(* Logix 5000 project; controller HPU_Part_Evac_Start 1769-L33ERM rev 30.11; software revision 30.01 *)

TASK MainTask (continuous, watchdog 500 ms) : MainProgram, Motion_Tools

MODULES
   Local : 1769-L33ERM (Compact 0, rev 30.11)
      Ecyl_1 : vendor 1 type 37 code 32 (Ethernet 192.168.1.21, rev 2.1, MotionSync RPI 1 ms, MotionDiagnostics RPI 1 ms)   // E Cylinder Station 1
      Ecyl_2 : vendor 1 type 37 code 32 (Ethernet 192.168.1.22, rev 2.1, MotionDiagnostics RPI 1 ms, MotionSync RPI 1 ms)   // E Cylinder Station 2
      Ecyl_4 : vendor 1 type 37 code 32 (Ethernet 192.168.1.24, rev 2.1, MotionSync RPI 1 ms, MotionDiagnostics RPI 1 ms)   // E Cylinder Station 4
      Ecyl_3 : vendor 1 type 37 code 32 (Ethernet 192.168.1.23, rev 2.1, MotionSync RPI 1 ms, MotionDiagnostics RPI 1 ms)   // E Cylinder Station 3
END_MODULES

TYPE Sequence1 :   // Sequence Start Conditions Met
STRUCT
   Perm : BOOL;   // Permissive to Advance
   Step : INT;   // Step Number
   Fault : BOOL;   // Fault
   Fault_Code : INT;   // Fault Code
   On : BOOL;   // Enabled
   StepMode : BOOL;   // Step Mode Enabled
   StepNext : BOOL;   // Next Step
   Status : STRING;   // Current Status
   Reset : BOOL;   // Reset Sequence
   Complete : BOOL;   // Sequence Complete [OS]
   PermLostStep : INT;   // Step where Permissive was Lost
   Home : BOOL;   // Sequence Actuators at Home
   StartCond : BOOL;   // Sequence Start Conditions Met
   HomeReq : BOOL;   // Sequence Home Request
   Step_Msg : STRING;   // Operator Message from Sequence
END_STRUCT
END_TYPE

TYPE Sequence_Ctrl :   // Sequence Start Conditions Met
STRUCT
   Perm : BOOL;   // Permissive to Advance
   Step : INT;   // Step Number
   Fault : BOOL;   // Fault
   Fault_Code : INT;   // Fault Code
   On : BOOL;   // Enabled
   StepMode : BOOL;   // Step Mode Enabled
   StepNext : BOOL;   // Next Step
   Status : STRING;   // Current Status
   Reset : BOOL;   // Reset Sequence
   Complete : BOOL;   // Sequence Complete [OS]
   PermLostStep : INT;   // Step where Permissive was Lost
   Home : BOOL;   // Sequence Actuators at Home
   StartCond : BOOL;   // Sequence Start Conditions Met
   HomeReq : BOOL;   // Sequence Home Request
   Step_Msg : STRING;   // Operator Message from Sequence
END_STRUCT
END_TYPE

VAR_GLOBAL   (* controller tags *)
   _Always_Off : BOOL;   // Always Off
   ai_Cylinder_Posn_Sta_1 : INT;   // Cylinder Position Station 1 Analog Input Raw Count Value
   ai_Cylinder_Posn_Sta_2 : INT;   // Cylinder Pressure Station 2 Analog Input Raw Count Value
   ai_Cylinder_Posn_Sta_3 : INT;   // Cylinder Pressure Station 3 Analog Input Raw Count Value
   ai_Cylinder_Posn_Sta_4 : INT;   // Cylinder Pressure Station 4 Analog Input Raw Count Value
   ai_Cylinder_Press_Sta_1 : INT;   // Cylinder Pressure Station 1 Analog Input Raw Count Value
   ai_Cylinder_Press_Sta_2 : INT;   // Cylinder Pressure Station 2 Analog Input Raw Count Value
   ai_Cylinder_Press_Sta_3 : INT;   // Cylinder Pressure Station 3 Analog Input Raw Count Value
   ai_Cylinder_Press_Sta_4 : INT;   // Cylinder Pressure Station 4 Analog Input Raw Count Value
   ao_Pressure_Relief_Out_Sta_1 : INT;   // Cylinder Relief Pressure Output Station 1 Analog Output Raw Count Value
   ao_Pressure_Relief_Out_Sta_2 : INT;   // Cylinder Relief Pressure Output Station 2 Analog Output Raw Count Value
   ao_Pressure_Relief_Out_Sta_3 : INT;   // Cylinder Relief Pressure Output Station 3 Analog Output Raw Count Value
   ao_Pressure_Relief_Out_Sta_4 : INT;   // Cylinder Relief Pressure Output Station 4 Analog Output Raw Count Value
   c_Ecyl_1_Auto_Exe_Inc : BOOL;   // Coil Ecylinder 1 Axis Auto Move (Incremental Move)
   c_MCR_On_Dly_PUL : BOOL;   // Coil MCR is On (1 Sec Delay) (250ms Pulse)
   c_Sld_Auto_Exe : BOOL;   // Coil Slide Auto Move (Absolute)
   c_Sld_Man_DS_Exe : BOOL;   // Coil Slide Axis Manual Move (Drive Screen)
   c_Sld_Man_PS_Cut : BOOL;   // Coil Slide Axis Manual Move Cut Position Pro Stich
   c_Sld_Man_PS_Grind : BOOL;   // Coil Slide Axis Manual Move Grind Position Pro Stich
   c_Sld_Man_PS_Grind_End : BOOL;   // Coil Slide Axis Manual Move Grind End Position Pro Stich
   c_Sld_Man_PS_Home : BOOL;   // Coil Slide Axis Manual Move Home Position Pro Stich
   c_Sld_Man_TR_End : BOOL;   // Coil Slide Axis Manual Move End Position Trheaded Rod
   c_Sld_Man_TR_Home : BOOL;   // Coil Slide Axis Manual Move Home Position Trheaded Rod
   c_Sld_Man_TR_Start : BOOL;   // Coil Slide Axis Manual Move Start Position Trheaded Rod
   c_Sld_Man_TR_Taper_Start : BOOL;   // Coil Slide Axis Manual Move Taper Start Position Trheaded Rod
   cntl_Mag_sld : MOTION_INSTRUCTION := (FLAGS := 570425344, DN := 1);   // Axes Sync Control
   cntl_Rot_UnSync : MOTION_INSTRUCTION := (FLAGS := 704643072, DN := 1, PC := 1);
   cntl_Sld_Air_Stop : MOTION_INSTRUCTION := (FLAGS := 33554432);
   cntl_Sld_Chng_Spd : MOTION_INSTRUCTION := (FLAGS := 570425344, DN := 1);
   cntl_Sld_Home : MOTION_INSTRUCTION := (FLAGS := 704643072, DN := 1, PC := 1, STATE := 17);   // Servo Control Slide Axis Home
   cntl_Sld_Off : MOTION_INSTRUCTION := (FLAGS := 570425344, DN := 1, STATUS := 2, STATE := 1);   // Servo Control Slide Axis Off
   cntl_Sld_On : MOTION_INSTRUCTION := (FLAGS := 570425344, DN := 1, STATE := 1);   // Servo Control Slide Axis On
   cntl_Sld_Reset : MOTION_INSTRUCTION := (FLAGS := 570425344, DN := 1, STATE := 1);   // Servo Control Slide Axis Fault Reset
   cntl_Sld_SD_Reset : MOTION_INSTRUCTION := (FLAGS := 33554432);   // Servo Control Slide Axis Shutdown Reset
   cntl_Sld_Stop : MOTION_INSTRUCTION := (FLAGS := 33554432);   // Motion Control Slide Axis Axis Stop
   cPV_Sld_Tpr_Vel : REAL := 0.033333335;   // Calculated slide velocity for tapered portion of thread.
   cPV_Sta_1_Cyl_Posn : REAL;   // Scaled Station 1 Stacking Cyclinder Position
   cPV_Sta_1_Cyl_Pressure : REAL;   // Scaled Station 1 Stacking Cyclinder Pressure
   cPV_Sta_2_Cyl_Posn : REAL;   // Scaled Station 2 Stacking Cyclinder Position
   cPV_Sta_2_Cyl_Pressure : REAL;   // Scaled Station 2 Stacking Cyclinder Position
   cPV_Sta_3_Cyl_Posn : REAL;   // Scaled Station 3 Stacking Cyclinder Position
   cPV_Sta_3_Cyl_Pressure : REAL;   // Scaled Station 3 Stacking Cyclinder Position
   cPV_Sta_4_Cyl_Posn : REAL;   // Scaled Station 4 Stacking Cyclinder Position
   cPV_Sta_4_Cyl_Pressure : REAL;   // Scaled Station 4 Stacking Cyclinder Position
   cSP_TR_Pitch : REAL := 5.0;   // Treaded Rod Pitch
   cSP_TR_Ratio : REAL := 1800.0;
   Drives_OK : BOOL := 1;   // All Drives OK
   ECyl_1 : AXIS_CIP_DRIVE;   // E Cylinder # 1
   ECyl_2 : AXIS_CIP_DRIVE;   // E Cylinder # 2
   Ecyl_3 : AXIS_CIP_DRIVE;
   Ecyl_4 : AXIS_CIP_DRIVE;
   hPB_All_Servo_On : BOOL;   // HMI Pushbutton All Servos On
   hPB_All_Servos_Off : BOOL;   // HMI Pushbutton All Servos OFF
   Hpb_Home : BOOL;   // HMI Pushbutton Machine Home
   hPB_MS_Hyd_Pump : BOOL;   // HMI PB Enable Hydraulic Pump
   hPB_Sld_AbsMv : BOOL;   // HMI Pushbutton Datum Bottom Axis Manual Move Absolute (From Drive Screen)
   hPB_Sld_Home : BOOL;   // HMI Pushbutton Slide Axis Home
   hPB_Sld_IncMv : BOOL;   // HMI Pushbutton Slide Axis Manual Move Incremental (From Drive Screen)
   hPB_Sld_MMv_PS_Cut : BOOL;   // HMI Pushbutton Slide Axis Pro Stich >>Move to Cut Position
   hPB_Sld_MMv_PS_Grind : BOOL;   // HMI Pushbutton Slide Axis Pro Stich >>Move to Grind Position
   hPB_Sld_MMv_PS_Grind_End : BOOL;   // HMI Pushbutton Slide Axis Pro Stich >>Move to Grind End Position
   hPB_Sld_MMv_PS_Home : BOOL;   // HMI Pushbutton Slide Axis Pro Stich >>Move to Home Position
   hPB_Sld_MMv_TR_End : BOOL;   // HMI Pushbutton Slide Axis Threaded Rod >>Move to End Position
   hPB_Sld_MMv_TR_Home : BOOL;   // HMI Pushbutton Slide Axis Threaded Rod >>Move to Home Position
   hPB_Sld_MMv_TR_Start : BOOL;   // HMI Pushbutton Slide Axis Threaded Rod >>Move to Start Position
   hPB_Sld_MMv_TR_Taper_Start : BOOL;   // HMI Pushbutton Slide Axis Threaded Rod >>Move to Taper Start Position
   hPB_Sld_Reset : BOOL;   // HMI Pushbutton Slide Axis Servo Reset
   hPB_Sld_ServoOff : BOOL;   // HMI Pushbutton Slide Axis Servo Axis Servo Off
   hPB_Sld_ServoOn : BOOL;   // HMI Pushbutton Slide Axis Servo Axis Servo On
   hPB_SV_Dump_Valve : BOOL;   // HMI PB Pressure Dump Solenoid Valve
   hPB_Sync_R_S : BOOL;   // Sync Rotary to Slide
   hPB_UnSync_R_S : BOOL;   // UnSync Rotary Axis from Slide
   hpl_Ecyl_1_Enabled : BOOL;   // E Cylinder 1 Enabled
   hpl_Ecyl_2_Enabled : BOOL;   // E Cylinder 2 Enabled
   hPL_PS_Active : BOOL;   // Pro-Stich Sequence Active
   hpv_Ecyl_1_Posn : REAL;   // E Cylinder 1 Position (mm)
   hpv_Ecyl_2_Posn : REAL;   // E Cylinder 2 Position (mm)
   hpv_Ecyl_3_Enabled : BOOL;   // E Cylinder 3 Enabled
   hpv_Ecyl_3_Posn : REAL;   // E Cylinder 3 Position (mm)
   hpv_Ecyl_4_Enabled : BOOL;   // E Cylinder 4 Enabled
   hpv_Ecyl_4_Posn : REAL;   // E Cylinder 4 Position (mm)
   hSP_Ecyl_1_DS_AbsMov : REAL := 10.0;   // HMI Setpoint Ecylinder 1 Axis (Drive Screen) Manual Absolute Move
   hSP_Ecyl_1_DS_IncMov : REAL := 20.0;   // HMI Setpoint Ecylinder 1 Axis (Drive Screen) Manual Incremental Move
   hSP_Ecyl_ManMove_Vel : REAL := 25.0;   // HMI Setpoint Ecylinder Axis Manual Move Velocity
   hSP_Ecyl_Pos_DB : REAL := 0.01;   // HMI Setpoint Ecylinder Positioning Deadband
   hSP_PS_Ecyl_1_Psp_Clear : REAL := 161.7784;   // HMI Setpoint Ecylinder 1 Clear of Stacking Cylinder Location
   hSP_PS_Ecyl_1_Psp_Home : REAL := 10.0;   // HMI Setpoint Ecylinder 1 HOME
   hSP_PS_Ecyl_1_Psp_Stacking : REAL := 166.4166;   // HMI Setpoint Ecylinder 1 Stacking Location
   hSP_PS_Ecyl_1_Psp_Unload : REAL := 158.5634;   // HMI Setpoint Ecylinder 1 Unload Location
   hSP_TR_Rot_Dir : DINT;
   hSP_TR_Sld_Psp_End : REAL := 100.0;   // Threaded Rod END Location Setpoint
   hSP_TR_Sld_Psp_Home : REAL := 10.0;   // Threaded Rod Home Position Setpoint
   hSP_TR_Sld_Psp_Start : REAL := 90.0;   // Threaded Rod START Position Setpoint
   hSP_TR_Sld_Psp_Taper_Start : REAL := 99.0;   // Threaded Rod Taper START Position Setpoint
   hSP_TR_TPM : REAL := 5.0;   // Treaded Rod Threads per Millimeter
   i_cr_Die_Position : BOOL;   // Die Position Sensor 1 = Die Closed
   i_cr_E_Stop : BOOL;   // Press Light Curtain and E Stop Input Relay Contacts
   i_cr_Pump_OL : BOOL;   // Hydraulic Pump Overload Contacts, NC
   i_cr_Pump_Running : BOOL;   // Hydraulic Pump running auxiliary contacts.
   i_cr_Stack_Done_Sta_1 : BOOL;   // Stack Done Station 1 signal from VAMCO
   i_cr_Stack_Done_Sta_2 : BOOL;   // Stack Done Station 2 signal from VAMCO
   i_cr_Stack_Done_Sta_3 : BOOL;   // Stack Done Station 3 signal from VAMCO
   i_cr_Stack_Done_Sta_4 : BOOL;   // Stack Done Station 4 signal from VAMCO
   i_pb_Cycle_Start : BOOL;   // Cycle Start Pushbutton Input
   i_pb_Cycle_Stop : BOOL;   // Cycle Stop Pushbutton Input
   i_pb_Reset : BOOL;   // Reset Pushbutton input
   IB_Man_Jog_Active : BOOL;   // Interface Bit used for Manual Jog Functions Starts Hydraulic Pump and Dump Valve
   IB_MS_Hyd_Pump : BOOL;   // Interface bit to run Hydraulic Pump in cycle.
   IB_PS_AMT_Sld : BOOL;   // Pro-Stich Auto Motion Trigger Slide Axis
   IB_PS_Loc_Ecyl_1_Clear : BOOL;   // Ecylinder 1 Location Bit Clear of Stacking Cylinder
   IB_PS_Loc_Ecyl_1_Home : BOOL := 1;   // Ecylinder 1 Location Bit Ecylinder 1 @ HOME
   IB_PS_Loc_Ecyl_1_Stacking : BOOL;   // Ecylinder 1 Location Bit Ecyl 1 @ Stacking
   IB_PS_Loc_Ecyl_1_Unload : BOOL;   // Ecylinder 1 Location Bit Ecylinder 1 @ Part Unload
   IB_SV_Dump_Valve : BOOL;   // Interface bit to trigger Dydraulic Pressure Dump Valve.
   IB_TR_AMT_Sld : BOOL;   // Threaded Rod Auto Motion Trigger Slide Axis
   IB_TR_Change_Speed : BOOL;   // Threaded Rod UnSync Axes
   IB_TR_Loc_Sld_End : BOOL;   // Threaded Rod Location Bit Slide @ END
   IB_TR_Loc_Sld_Home : BOOL := 1;   // Threaded Rod Location Bit Slide @ HOME
   IB_TR_Loc_Sld_Start : BOOL;   // Threaded Rod Location Bit Slide @ START
   IB_TR_Loc_Sld_Taper_Region : BOOL;   // Threaded Rod Location Bit Slide between Taper Start and END positions
   IB_TR_Loc_Sld_Taper_Start : BOOL;   // Threaded Rod Location Bit Slide at Taper Start position
   IB_TR_Sync_Axes : BOOL;   // Threaded Rod Sync Axes (Slave Rotate to Slide)
   IB_TR_UnSync_Axes : BOOL;   // Threaded Rod UnSync Axes
   M_Auto : BOOL;   // Machine in Auto Mode Sequence Cycle Start/Stop Active
   M_Manual : BOOL;   // Machine in Manual Mode, Outputs Controlled by HMI Buttons.
   M_Reset_Sum : BOOL;   // Machine Mode Reset_Sum
   MC_Sld_MAM : MOTION_INSTRUCTION := (FLAGS := 704643072, DN := 1, PC := 1);   // Motion Control Tag Slide Axis Motion Axis Move
   o_cr_Top_Stop : BOOL;   // Top Stop Relay Contacts to Press
   o_ms_Pump_Contactor : BOOL;   // Hydraulic Pump Contactor
   o_pl_Reset_Light : BOOL;   // Reset Pushbutton Light
   o_sv_Extend_Cyl_Sta_1 : BOOL;   // Extend Cylinder Station 1 Solenoid Valve
   o_sv_Extend_Cyl_Sta_2 : BOOL;   // Extend Cylinder Station 2 Solenoid Valve
   o_sv_Extend_Cyl_Sta_3 : BOOL;   // Extend Cylinder Station 3 Solenoid Valve
   o_sv_Extend_Cyl_Sta_4 : BOOL;   // Extend Cylinder Station 4 Solenoid Valve
   o_sv_Low_Press_Relief_Sta_1 : BOOL;   // Low Pressure Relief Diverter Station 1 Solenoid Valve
   o_sv_Low_Press_Relief_Sta_2 : BOOL;   // Low Pressure Relief Diverter Station 2 Solenoid Valve
   o_sv_Low_Press_Relief_Sta_3 : BOOL;   // Low Pressure Relief Diverter Station 3 Solenoid Valve
   o_sv_Low_Press_Relief_Sta_4 : BOOL;   // Low Pressure Relief Diverter Station 4 Solenoid Valve
   o_sv_Pressure_Dump : BOOL;   // Hydraulic Pressure Dump Valve
   o_sv_Retract_Cyl_Sta_1 : BOOL;   // Retract Cylinder Station 1 Solenoid Valve
   o_sv_Retract_Cyl_Sta_2 : BOOL;   // Retract Cylinder Station 2 Solenoid Valve
   o_sv_Retract_Cyl_Sta_3 : BOOL;   // Retract Cylinder Station 3 Solenoid Valve
   o_sv_Retract_Cyl_Sta_4 : BOOL;   // Retract Cylinder Station 4 Solenoid Valve
   ons_Sld_003 : BOOL;
   p_Ecyl_1 : BOOL := 1;   // Permissive (for Movement) Ecylinder 1 Axis
   p_hyd_dump_vlv : BOOL;
   p_hyd_pump : BOOL;
   Seq_ProStch : Sequence1 := (Step_Msg := 'Rotary Stopped');   // Pro-Stich, Synthes Sequence
   Seq_ThdRd : Sequence1 := (Home := 1, Step_Msg := 'Slide @ Home Location');
   SP_Ecyl_1_Move_Type : DINT;   // Move Type Ecylinder 1 0=Absolute 1=Incremental
   SP_Ecyl_1_Pos : REAL := 10.0;   // Setpoint Ecylinder 1 Axis Position (Used in MAM)
   SP_Ecyl_1_Vel : REAL := 100.0;   // Setpoint Ecyl 1 Axis Velocity
   Station_1 : MOTION_GROUP;
   z_Slide_Pos_Buff : REAL := 443.1691;
   z_stop_sld : BOOL;
   z_test_002 : BOOL;
END_VAR

PROGRAM MainProgram   (* main routine MainRoutine *)

ROUTINE MainRoutine   (* ladder *)
END_ROUTINE

ROUTINE r1_Analog_IO   (* ladder *)
// Analog Conversions, scaling, etc.
   0: ;
END_ROUTINE

ROUTINE r2_Outputs   (* ladder *)
// Digital Output Control
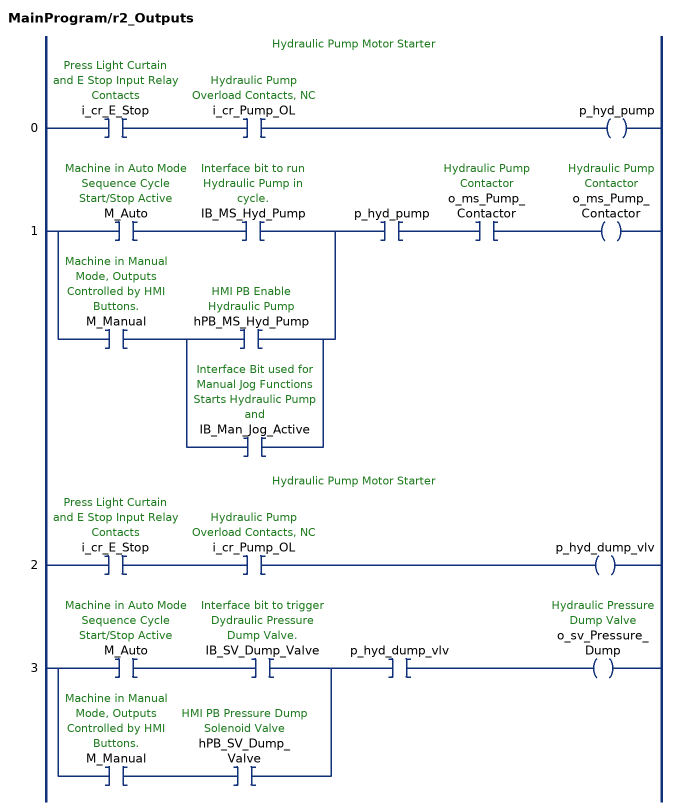
   // Hydraulic Pump Motor Starter
   0: XIC(i_cr_E_Stop)XIC(i_cr_Pump_OL)OTE(p_hyd_pump);
   1: [XIC(M_Auto) XIC(IB_MS_Hyd_Pump) ,XIC(M_Manual) [XIC(hPB_MS_Hyd_Pump) ,XIC(IB_Man_Jog_Active) ] ]XIC(p_hyd_pump)XIC(o_ms_Pump_Contactor)OTE(o_ms_Pump_Contactor);
   // Hydraulic Pump Motor Starter
   2: XIC(i_cr_E_Stop)XIC(i_cr_Pump_OL)OTE(p_hyd_dump_vlv);
   3: [XIC(M_Auto) XIC(IB_SV_Dump_Valve) ,XIC(M_Manual) XIC(hPB_SV_Dump_Valve) ]XIC(p_hyd_dump_vlv)OTE(o_sv_Pressure_Dump);
END_ROUTINE
END_PROGRAM

PROGRAM Motion_Tools
VAR
   cSld_ESR_MT : BOOL;   // Slide Axis E-Stop Recovery Motion Trigger [OS]
   cSld_EStp : BOOL;   // Slide Axis Has been Stopped on E-Stop Condition
   cSld_IM_Estp : BOOL;   // Interface Bit Slide Axis E-Stop While in Motion [OS]
   ons_Sld_001 : BOOL;
   ons_Sld_002 : BOOL;
END_VAR

ROUTINE r1_Ecyl_1   (* ladder *)
// Ecylinder 1 Axis
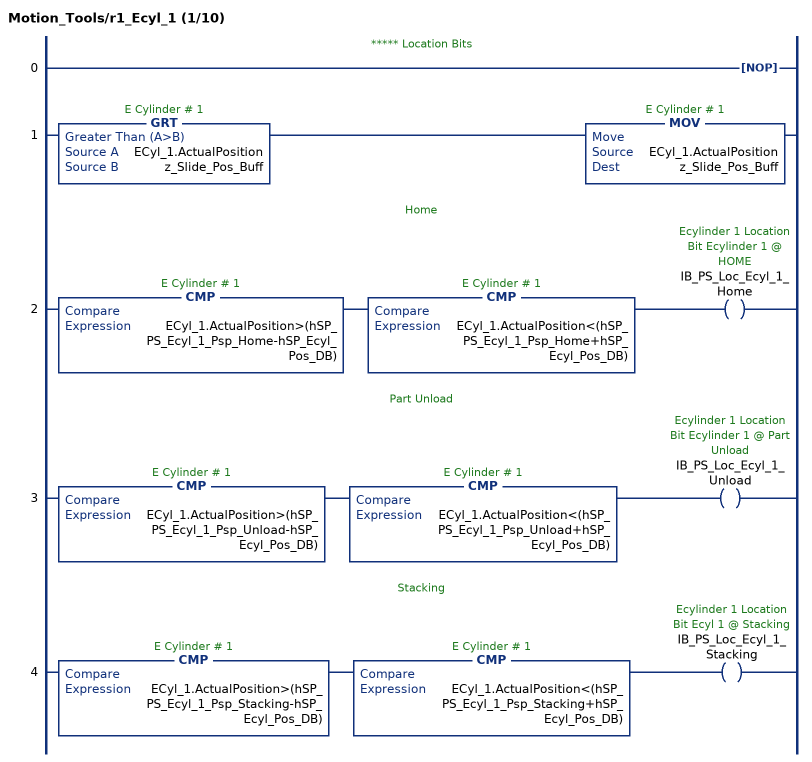
   // ***** Location Bits
   0: NOP();
   1: GRT(ECyl_1.ActualPosition,z_Slide_Pos_Buff)MOV(ECyl_1.ActualPosition,z_Slide_Pos_Buff);
   // Home
   2: CMP(ECyl_1.ActualPosition>(hSP_PS_Ecyl_1_Psp_Home-hSP_Ecyl_Pos_DB))CMP(ECyl_1.ActualPosition<(hSP_PS_Ecyl_1_Psp_Home+hSP_Ecyl_Pos_DB))OTE(IB_PS_Loc_Ecyl_1_Home);
   // Part Unload
   3: CMP(ECyl_1.ActualPosition>(hSP_PS_Ecyl_1_Psp_Unload-hSP_Ecyl_Pos_DB))CMP(ECyl_1.ActualPosition<(hSP_PS_Ecyl_1_Psp_Unload+hSP_Ecyl_Pos_DB))OTE(IB_PS_Loc_Ecyl_1_Unload);
   // Stacking
   4: CMP(ECyl_1.ActualPosition>(hSP_PS_Ecyl_1_Psp_Stacking-hSP_Ecyl_Pos_DB))CMP(ECyl_1.ActualPosition<(hSP_PS_Ecyl_1_Psp_Stacking+hSP_Ecyl_Pos_DB))OTE(IB_PS_Loc_Ecyl_1_Stacking);
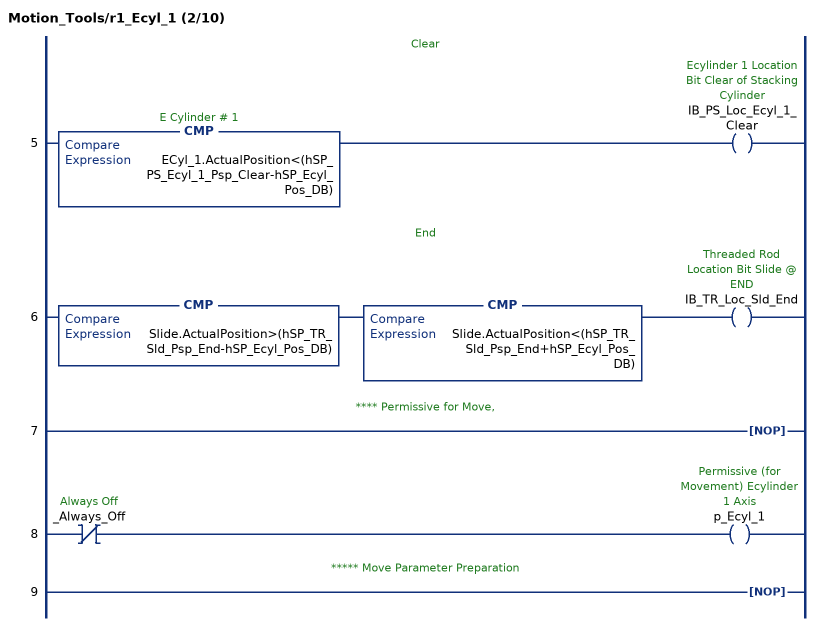
   // Clear
   5: CMP(ECyl_1.ActualPosition<(hSP_PS_Ecyl_1_Psp_Clear-hSP_Ecyl_Pos_DB))OTE(IB_PS_Loc_Ecyl_1_Clear);
   // End
   6: CMP(Slide.ActualPosition>(hSP_TR_Sld_Psp_End-hSP_Ecyl_Pos_DB))CMP(Slide.ActualPosition<(hSP_TR_Sld_Psp_End+hSP_Ecyl_Pos_DB))OTE(IB_TR_Loc_Sld_End);
   // **** Permissive for Move,
   7: NOP();
   8: XIO(_Always_Off)OTE(p_Ecyl_1);
   // ***** Move Parameter Preparation
   9: NOP();
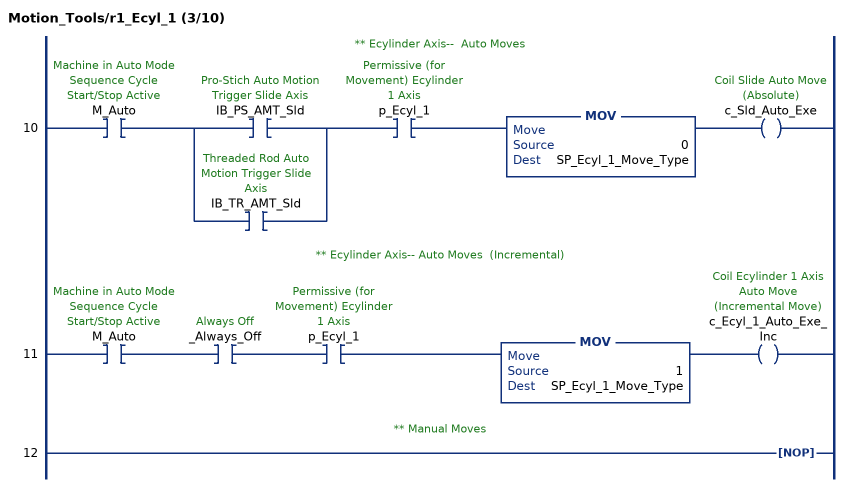
   // ** Ecylinder Axis--  Auto Moves
   10: XIC(M_Auto)[XIC(IB_PS_AMT_Sld) ,XIC(IB_TR_AMT_Sld) ]XIC(p_Ecyl_1)MOV(0,SP_Ecyl_1_Move_Type)OTE(c_Sld_Auto_Exe);
   // ** Ecylinder Axis-- Auto Moves  (Incremental)
   11: XIC(M_Auto)XIC(_Always_Off)XIC(p_Ecyl_1)MOV(1,SP_Ecyl_1_Move_Type)OTE(c_Ecyl_1_Auto_Exe_Inc);
   // ** Manual Moves
   12: NOP();
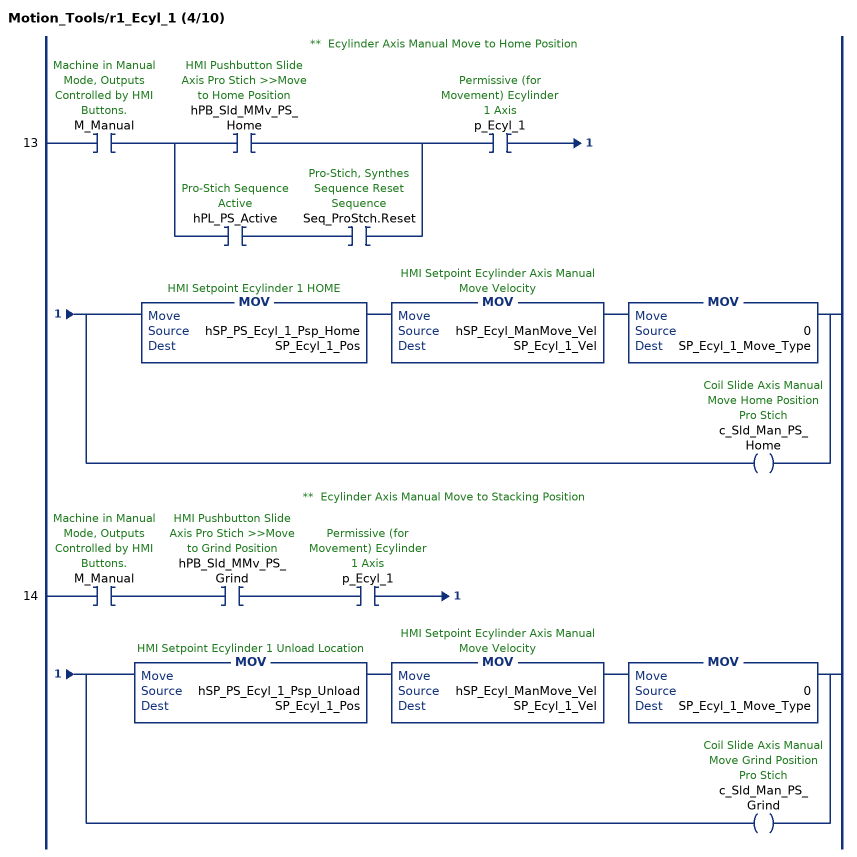
   // **  Ecylinder Axis Manual Move to Home Position
   13: XIC(M_Manual)[XIC(hPB_Sld_MMv_PS_Home) ,XIC(hPL_PS_Active) XIC(Seq_ProStch.Reset) ]XIC(p_Ecyl_1)[MOV(hSP_PS_Ecyl_1_Psp_Home,SP_Ecyl_1_Pos) MOV(hSP_Ecyl_ManMove_Vel,SP_Ecyl_1_Vel) MOV(0,SP_Ecyl_1_Move_Type) ,OTE(c_Sld_Man_PS_Home) ];
   // **  Ecylinder Axis Manual Move to Stacking Position
   14: XIC(M_Manual)XIC(hPB_Sld_MMv_PS_Grind)XIC(p_Ecyl_1)[MOV(hSP_PS_Ecyl_1_Psp_Unload,SP_Ecyl_1_Pos) MOV(hSP_Ecyl_ManMove_Vel,SP_Ecyl_1_Vel) MOV(0,SP_Ecyl_1_Move_Type) ,OTE(c_Sld_Man_PS_Grind) ];
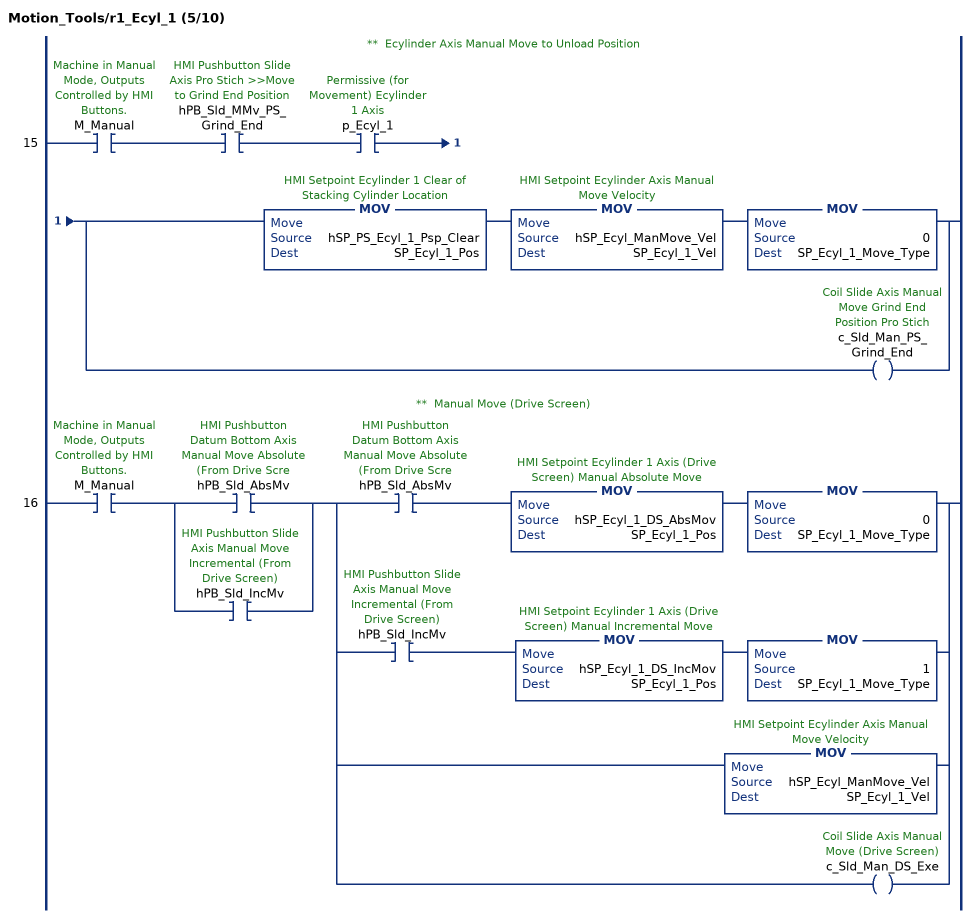
   // **  Ecylinder Axis Manual Move to Unload Position
   15: XIC(M_Manual)XIC(hPB_Sld_MMv_PS_Grind_End)XIC(p_Ecyl_1)[MOV(hSP_PS_Ecyl_1_Psp_Clear,SP_Ecyl_1_Pos) MOV(hSP_Ecyl_ManMove_Vel,SP_Ecyl_1_Vel) MOV(0,SP_Ecyl_1_Move_Type) ,OTE(c_Sld_Man_PS_Grind_End) ];
   // **  Manual Move (Drive Screen)
   16: XIC(M_Manual)[XIC(hPB_Sld_AbsMv) ,XIC(hPB_Sld_IncMv) ][[XIC(hPB_Sld_AbsMv) MOV(hSP_Ecyl_1_DS_AbsMov,SP_Ecyl_1_Pos) MOV(0,SP_Ecyl_1_Move_Type) ,XIC(hPB_Sld_IncMv) MOV(hSP_Ecyl_1_DS_IncMov,SP_Ecyl_1_Pos) MOV(1,SP_Ecyl_1_Move_Type) ] ,MOV(hSP_Ecyl_ManMove_Vel,SP_Ecyl_1_Vel) ,OTE(c_Sld_Man_DS_Exe) ];
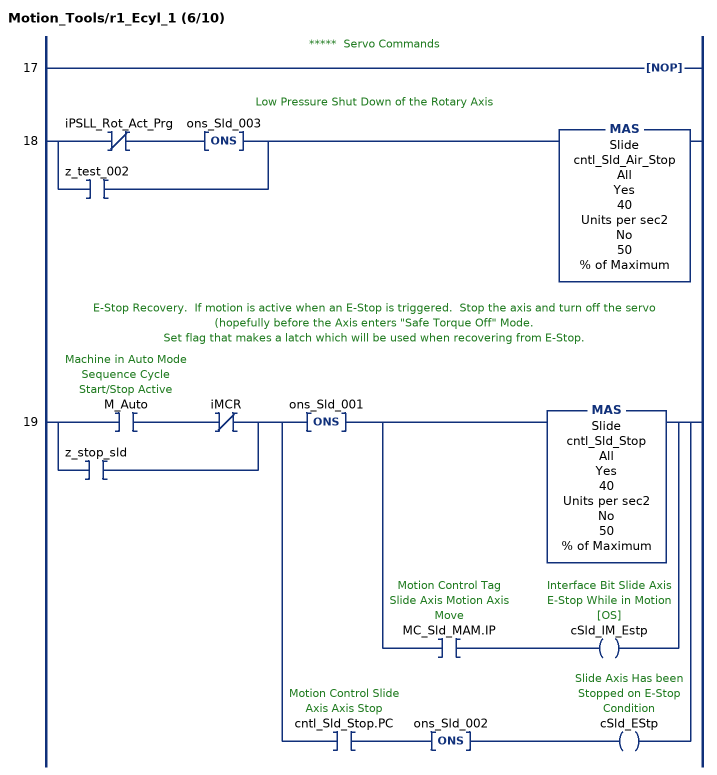
   // *****  Servo Commands
   17: NOP();
   // Low Pressure Shut Down of the Rotary Axis
   18: [XIO(iPSLL_Rot_Act_Prg) ONS(ons_Sld_003) ,XIC(z_test_002) ]MAS(Slide,cntl_Sld_Air_Stop,All,Yes,40,Units per sec2,No,50,% of Maximum);
   // E-Stop Recovery.  If motion is active when an E-Stop is triggered.  Stop the axis and turn off the servo (hopefully before the Axis enters "Safe Torque Off" Mode.
   // Set flag that makes a latch which will be used when recovering from E-Stop.
   19: [XIC(M_Auto) XIO(iMCR) ,XIC(z_stop_sld) ][ONS(ons_Sld_001) [MAS(Slide,cntl_Sld_Stop,All,Yes,40,Units per sec2,No,50,% of Maximum) ,XIC(MC_Sld_MAM.IP) OTE(cSld_IM_Estp) ] ,XIC(cntl_Sld_Stop.PC) ONS(ons_Sld_002) OTE(cSld_EStp) ];
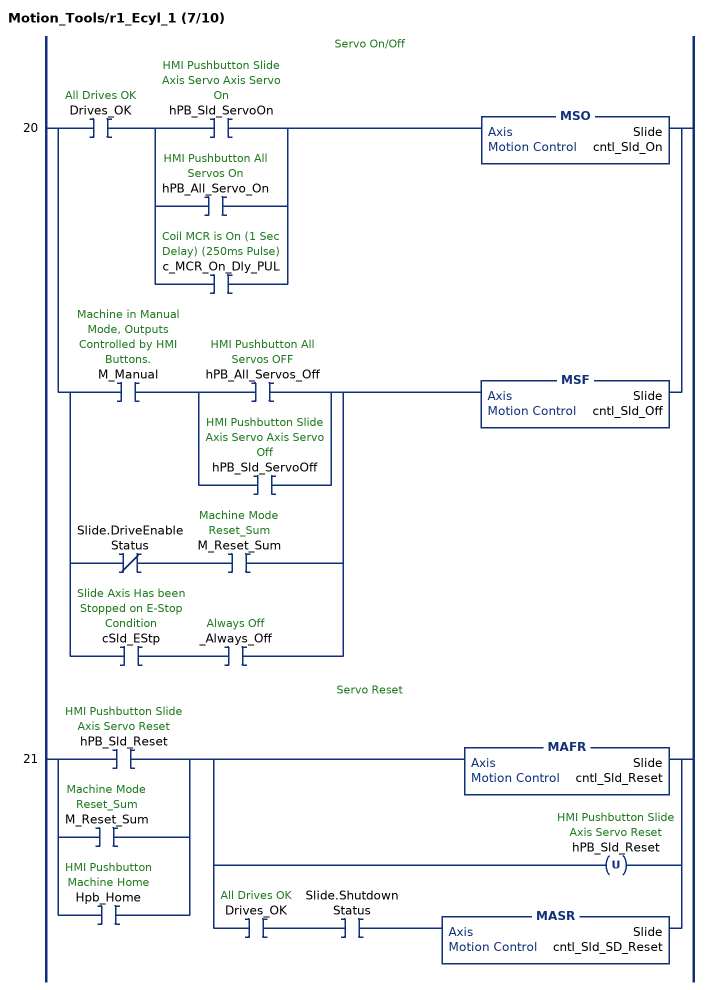
   // Servo On/Off
   20: [XIC(Drives_OK) [XIC(hPB_Sld_ServoOn) ,XIC(hPB_All_Servo_On) ,XIC(c_MCR_On_Dly_PUL) ] MSO(Slide,cntl_Sld_On) ,[XIC(M_Manual) [XIC(hPB_All_Servos_Off) ,XIC(hPB_Sld_ServoOff) ] ,XIO(Slide.DriveEnableStatus) XIC(M_Reset_Sum) ,XIC(cSld_EStp) XIC(_Always_Off) ] MSF(Slide,cntl_Sld_Off) ];
   // Servo Reset
   21: [XIC(hPB_Sld_Reset) ,XIC(M_Reset_Sum) ,XIC(Hpb_Home) ][[MAFR(Slide,cntl_Sld_Reset) ,OTU(hPB_Sld_Reset) ] ,XIC(Drives_OK) XIC(Slide.ShutdownStatus) MASR(Slide,cntl_Sld_SD_Reset) ];
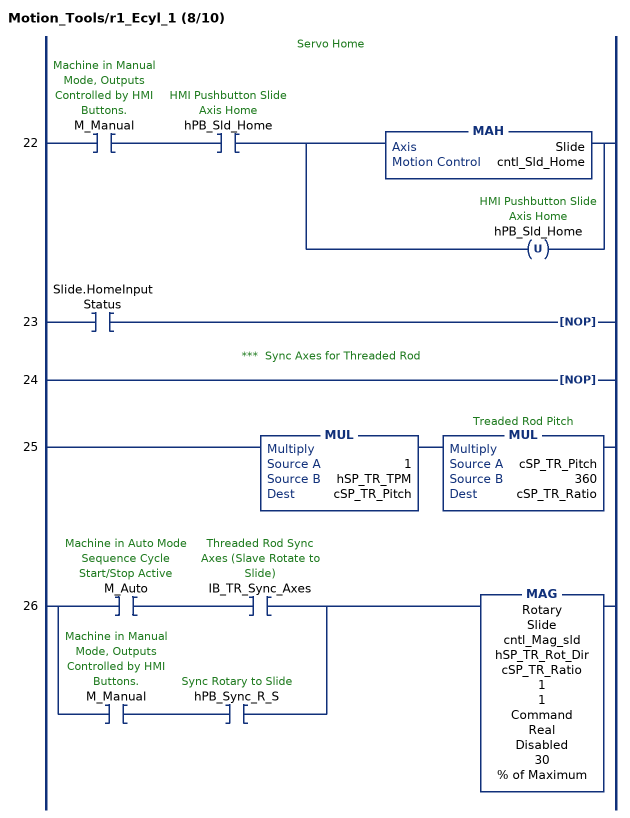
   // Servo Home
   22: XIC(M_Manual)XIC(hPB_Sld_Home)[MAH(Slide,cntl_Sld_Home) ,OTU(hPB_Sld_Home) ];
   23: XIC(Slide.HomeInputStatus)NOP();
   // ***  Sync Axes for Threaded Rod
   24: NOP();
   25: MUL(1,hSP_TR_TPM,cSP_TR_Pitch)MUL(cSP_TR_Pitch,360,cSP_TR_Ratio);
   26: [XIC(M_Auto) XIC(IB_TR_Sync_Axes) ,XIC(M_Manual) XIC(hPB_Sync_R_S) ]MAG(Rotary,Slide,cntl_Mag_sld,hSP_TR_Rot_Dir,cSP_TR_Ratio,1,1,Command,Real,Disabled,30,% of Maximum);
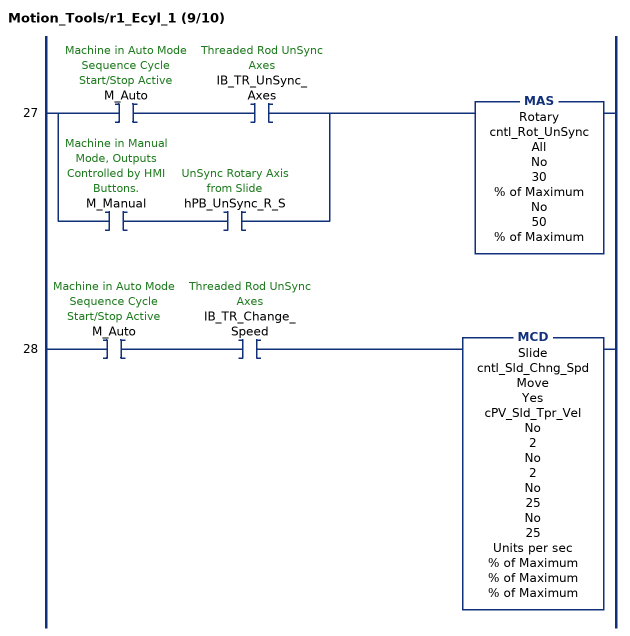
   27: [XIC(M_Auto) XIC(IB_TR_UnSync_Axes) ,XIC(M_Manual) XIC(hPB_UnSync_R_S) ]MAS(Rotary,cntl_Rot_UnSync,All,No,30,% of Maximum,No,50,% of Maximum);
   28: XIC(M_Auto)XIC(IB_TR_Change_Speed)MCD(Slide,cntl_Sld_Chng_Spd,Move,Yes,cPV_Sld_Tpr_Vel,No,2,No,2,No,25,No,25,Units per sec,% of Maximum,% of Maximum,% of Maximum);
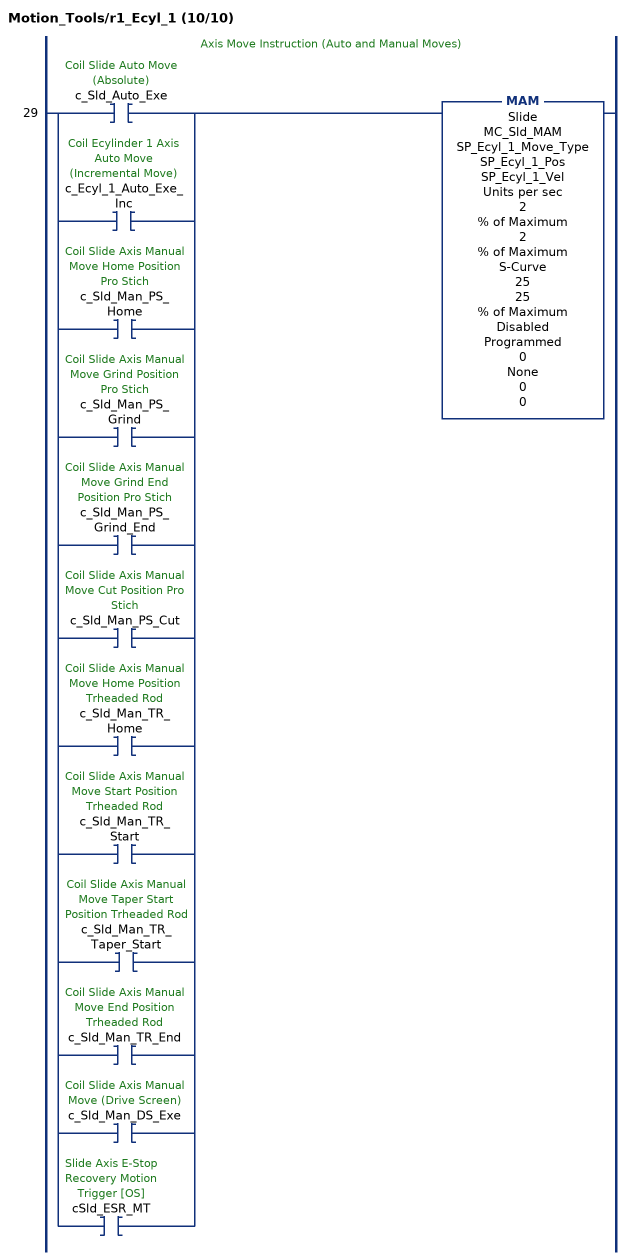
   // Axis Move Instruction (Auto and Manual Moves)
   29: [XIC(c_Sld_Auto_Exe) ,XIC(c_Ecyl_1_Auto_Exe_Inc) ,XIC(c_Sld_Man_PS_Home) ,XIC(c_Sld_Man_PS_Grind) ,XIC(c_Sld_Man_PS_Grind_End) ,XIC(c_Sld_Man_PS_Cut) ,XIC(c_Sld_Man_TR_Home) ,XIC(c_Sld_Man_TR_Start) ,XIC(c_Sld_Man_TR_Taper_Start) ,XIC(c_Sld_Man_TR_End) ,XIC(c_Sld_Man_DS_Exe) ,XIC(cSld_ESR_MT) ]MAM(Slide,MC_Sld_MAM,SP_Ecyl_1_Move_Type,SP_Ecyl_1_Pos,SP_Ecyl_1_Vel,Units per sec,2,% of Maximum,2,% of Maximum,S-Curve,25,25,% of Maximum,Disabled,Programmed,0,None,0,0);
END_ROUTINE
END_PROGRAM
